PROGRAM MAIN
VAR
	RobotWorkcenterControl			:		RobotWorkcenterControl;
	RobotSimulation					:		RobotSimulation;
	WorkcenterSimulation			:		WorkcenterSimulation;
	
	Start							: 		BOOL;
END_VAR
VAR // added by the converter: edge detectors and wires of the graphical bodies
    _w1 : BOOL;
END_VAR

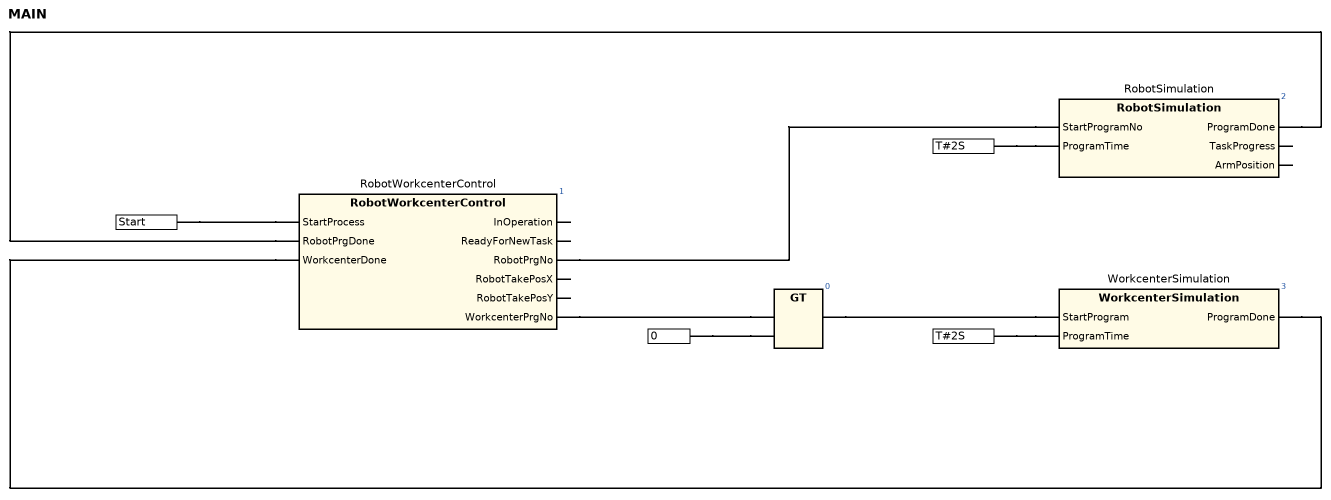
_w1 := RobotWorkcenterControl.WorkcenterPrgNo > 0;
RobotWorkcenterControl(
    StartProcess := Start,
    RobotPrgDone := RobotSimulation.ProgramDone,
    WorkcenterDone := WorkcenterSimulation.ProgramDone);
RobotSimulation(StartProgramNo := RobotWorkcenterControl.RobotPrgNo, ProgramTime := T#2S);
WorkcenterSimulation(StartProgram := _w1, ProgramTime := T#2S);

END_PROGRAM

(* stored: Version 1.1.0.1, ProductVersion 3.1.4024.15
   POU MAIN: Id {08b88ad3-29ba-486e-82aa-dc7f55bdebbc}, SpecialFunc None *)
